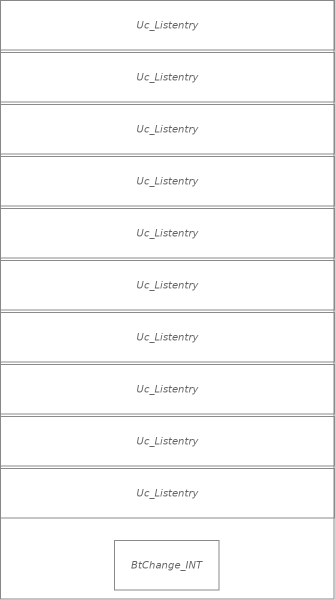
VISUALIZATION Uc_List  // 335x600
    Frame (0,0 335x50)
        shows Uc_Listentry(nId := nIdStartpoint+ 0, stVisu := stVisu)
    Frame (0,52 335x50)
        shows Uc_Listentry(nId := nIdStartpoint+ 1, stVisu := stVisu)
    Frame (0,104 335x50)
        shows Uc_Listentry(nId := nIdStartpoint+ 2, stVisu := stVisu)
    Frame (0,156 335x50)
        shows Uc_Listentry(nId := nIdStartpoint+ 3, stVisu := stVisu)
    Frame (0,208 335x50)
        shows Uc_Listentry(nId := nIdStartpoint+ 4, stVisu := stVisu)
    Frame (0,260 335x50)
        shows Uc_Listentry(nId := nIdStartpoint+ 5, stVisu := stVisu)
    Frame (0,312 335x50)
        shows Uc_Listentry(nId := nIdStartpoint+ 6, stVisu := stVisu)
    Frame (0,364 335x50)
        shows Uc_Listentry(nId := nIdStartpoint+ 7, stVisu := stVisu)
    Frame (0,416 335x50)
        shows Uc_Listentry(nId := nIdStartpoint+ 8, stVisu := stVisu)
    Frame (0,468 335x50)
        shows Uc_Listentry(nId := nIdStartpoint+ 9, stVisu := stVisu)
    Frame (114,540 105x50)
        shows BtChange_INT(Value := nIdStartpoint, minValue := 0, maxValue := 200, stepWidth := 1)
END_VISUALIZATION

(* stored: Version 1.1.0.1
   Visu Uc_List: Id {47da2968-ddab-43b6-8c7d-7f720b21e811} *)
